// TwinCAT 3 PLC project HOMS_XRT_PLC
// ProjectVersion: 1.0.0
// ProgramVersion: 3.1.4020.4
// libraries:
//   PMPS, * (SLAC - LCLS)
//   Tc2_ControllerToolbox, * (Beckhoff Automation GmbH)
//   Tc2_EtherCAT, * (Beckhoff Automation GmbH)
//   Tc2_MC2, * (Beckhoff Automation GmbH)
//   Tc2_Standard, * (Beckhoff Automation GmbH)
//   Tc2_System, * (Beckhoff Automation GmbH)
//   Tc2_Utilities, * (Beckhoff Automation GmbH)
//   Tc3_Module, * (Beckhoff Automation GmbH)
//   VisuDialogs, * (System)
//   LCLS General,2.4.2,SLAC
//   lcls-twincat-motion,1.4.2,SLAC
//   lcls-twincat-optics,0.1.1,SLAC
//   Tc2_SerialCom,3.3.7.0,Beckhoff Automation GmbH
// project tree:
//   Common/DUTs/ E_GantryControl.TcDUT (not stored), E_GantryMode.TcDUT (not stored), HOMS_Gantry.TcDUT (not stored), HOMS_GantryAxis.TcDUT (not stored), HOMS_PitchMechanismOld.TcDUT (not stored), ST_AbstractAxis.TcDUT (not stored), ST_CoEIndSub.TcDUT (not stored), ST_DecoupledMotionPermits.TcDUT (not stored), ST_ElmoGDCBellCoEParams.TcDUT (not stored), ST_HOMSStepper.TcDUT (not stored), ST_PiezoAxisOld.TcDUT (not stored), ST_StepperStatus.TcDUT (not stored)
//   Common/POUs/Helpers/ FB_Drive.TcPOU (not stored), FB_ElmoGDCBellCoE.TcPOU (not stored), FB_ElmoMCUploadDriveParams.TcPOU (not stored), FB_ElmoStoMonitor.TcPOU (not stored), FB_GantryDiffVirtualLimitSwitch.TcPOU (not stored), FB_InitDriveRefs.TcPOU (not stored), FB_LimitSwitchState.TcPOU (not stored), FB_PitchSoftLimits.TcPOU, FB_PI_E621_SerialDriver.TcPOU (not stored), FB_PI_E621_SerialTransaction.TcPOU (not stored), FB_PTP.TcPOU (not stored), FB_ReadFloatParameter.TcPOU (not stored), FB_ReadParameterInNC.TcPOU (not stored), FB_WriteParameterInNC.TcPOU (not stored), F_PiezoPosition.TcPOU (not stored), MC_SmoothMover.TcPOU (not stored), WithinRange.TcPOU (not stored)
//   Common/POUs/HOMS_FBs/ FB_Gantry.TcPOU (not stored), FB_GantryDifferenceMonitor.TcPOU (not stored), FB_PitchControlOld.TcPOU, FB_ReduceGantryDiff.TcPOU (not stored)
//   / GlobalTextList.TcGTLO (not stored), PiezoDriver.TcTTO (not stored), PlcTask.TcTTO (not stored), SerialIO.TcTTO (not stored), Visualization Manager.TcVMO (not stored)
//   GVLs/ GVL.TcGVL, GVL_COM_Buffers.TcGVL (not stored), GVL_Constants.TcGVL (not stored), GVL_Devices.TcGVL, GVL_IO.TcGVL (not stored), GVL_PMPS.TcGVL (not stored), GVL_SerialIO.TcGVL (not stored), GVL_XRTM1.TcGVL
//   POUs/ FB_MirrorCoatingProtection.TcPOU (not stored), FB_MirrorCoatingProtectionScaledPositions.TcPOU (not stored), FB_MPS_STATES.TcPOU (not stored), Main.TcPOU, PRG_CoatingProtectionScaledPositions.TcPOU (not stored), PRG_CoatingProtection.TcPOU, P_GantryDiffSup.TcPOU (not stored), P_MotionSup.TcPOU (not stored)
//   POUs/Modbus/ p_ModbusRx_OutputCoils.TcPOU (not stored), p_ModbusRx_PLCMemory.TcPOU, p_ModbusTx_InputCoils.TcPOU (not stored), p_ModbusTx_InputReg.TcPOU (not stored), p_ModbusTx_OutputCoils.TcPOU (not stored), p_ModbusTx_PLCMemory.TcPOU
//   POUs/Serial Comm/ PiezoSerial.TcPOU, P_Serial_Com.TcPOU (not stored)
//   VISUs/ GantryControls.TcVIS (not stored), Visualization.TcVIS (not stored), PiezoControls.TcVIS (not stored)
// real-time tasks:
//   TASK PlcTask: cycle T#10ms, priority 20, ADS port 350
//   TASK SerialIO: cycle T#2ms, priority 1, ADS port 351
//   TASK LoggerTask: cycle T#10ms, priority 2, ADS port 352
//   TASK PiezoDriver: cycle T#1ms, priority 3, ADS port 353
// motion (NC):
// I/O:
//   DEVICE HOMS, AmsNetId 172.21.88.136.2.1
//     Term 1 (EK1200) [EK1200-5000 EtherCAT Power supply (2A E-Bus)]
//       Term 24 (EL9187) [EL9187 Potential Connection, 8 x Ground]
//       Term 13 (EL2008) [EL2008 8Ch. Dig. Output 24V, 0.5A]
//       Term 14 (EK1122) [EK1122 2 port EtherCAT junction]
//         EK1100_M1 [EK1100 EtherCAT Coupler (2A E-Bus)]
//           EL7041-1000_M1_Xup [EL7041-1000 1Ch. Stepper motor output stage (50V, 5A, standard)]
//           EL7041-1000_M1_Xdwn [EL7041-1000 1Ch. Stepper motor output stage (50V, 5A, standard)]
//           EL7041-1000_M1_Yup [EL7041-1000 1Ch. Stepper motor output stage (50V, 5A, standard)]
//           EL7041-1000_M1_Ydwn [EL7041-1000 1Ch. Stepper motor output stage (50V, 5A, standard)]
//           EL7041-1000_M1_PitchCoarse [EL7041-1000 1Ch. Stepper motor output stage (50V, 5A, standard)]
//           EL7041-1000_M1_Bender
//           EL6001_M1_PitchFine [EL6001 Interface (RS232)]
//           EL5042_M1_Xupdwn
//           EL5042_M1_Yupdwn
//           EL5042_M1_PitchBender
//           EL1004_M1_STO
//           EL9505_M1_BenderLims
//           Term 42 (EL9011)
//         M2-Y1 (Elmo Drive) [Gold EtherCAT GCON Drive Rev:0x00010420]
//         M2-Y2 (Elmo Drive) [Gold EtherCAT GCON Drive Rev:0x00010420]
//         M2-X1 (Elmo Drive) [Gold EtherCAT GCON Drive Rev:0x00010420]
//         M2-X2 (Elmo Drive) [Gold EtherCAT GCON Drive Rev:0x00010420]
//         M2-P1 (Elmo Drive) [Gold EtherCAT GCON Drive Rev:0x00010420]
//         M2-B1 (Elmo Drive) [Gold EtherCAT GCON Drive Rev:0x00010420]
//         M2-Interface Box (EK1100) [EK1100 EtherCAT Coupler (2A E-Bus)]
//           M2-P1-Piezo (EL6001) [EL6001 Interface (RS232)]
//           M2 (EL9011) [EL9011 End Terminal]
//       Term 2 (EK1122) [EK1122 2 port EtherCAT junction]
//         M3-Y1 (Elmo Drive) [Gold EtherCAT GCON Drive Rev:0x00010420]
//         M3-Y2 (Elmo Drive) [Gold EtherCAT GCON Drive Rev:0x00010420]
//         M3-X1 (Elmo Drive) [Gold EtherCAT GCON Drive Rev:0x00010420]
//         M3-X2 (Elmo Drive) [Gold EtherCAT GCON Drive Rev:0x00010420]
//         M3-P1 (Elmo Drive) [Gold EtherCAT GCON Drive Rev:0x00010420]
//         M3-B1 (Elmo Drive) [Gold EtherCAT GCON Drive Rev:0x00010420]
//         M3-Interface Box (EK1100) [EK1100 EtherCAT Coupler (2A E-Bus)]
//           M3-P1-Piezo (EL6001) [EL6001 Interface (RS232)]
//           M3 (EL9011) [EL9011 End Terminal]
//       Term 34 (EK1521-0010)
// variable links:
//   HOMS_XRT_PLC Instance <-> HOMS
//     PlcTask Inputs/GVL.gAmsNetIDEcatMaster1 <-> InfoData/AmsNetId
//   HOMS_XRT_PLC Instance <-> HOMS/Term 1 (EK1200)/Term 13 (EL2008)
//     PlcTask Outputs/GVL.bXRT_M2_IN <-> Channel 2/Output
//     PlcTask Outputs/GVL.bXRT_M2_OUT <-> Channel 1/Output
//   HOMS_XRT_PLC Instance <-> HOMS/Term 1 (EK1200)/Term 14 (EK1122)/EK1100_M1/EL1004_M1_STO
//     PlcTask Inputs/Main.XRTM1.fbRunHOMS.bSTOEnable1 <-> Channel 1/Input
//     PlcTask Inputs/Main.XRTM1.fbRunHOMS.bSTOEnable2 <-> Channel 2/Input
//   HOMS_XRT_PLC Instance <-> HOMS/Term 1 (EK1200)/Term 14 (EK1122)/EK1100_M1/EL5042_M1_PitchBender
//     PlcTask Inputs/GVL_XRTM1.XRTM1_Pitch.diEncCnt <-> FB Inputs Channel 1/Position
//   HOMS_XRT_PLC Instance <-> HOMS/Term 1 (EK1200)/Term 14 (EK1122)/EK1100_M1/EL5042_M1_Xupdwn
//     PlcTask Inputs/Main.XRTM1.fbRunHOMS.stXdwnEnc/Count <-> FB Inputs Channel 2/Position
//     PlcTask Inputs/Main.XRTM1.fbRunHOMS.stXupEnc/Count <-> FB Inputs Channel 1/Position
//   HOMS_XRT_PLC Instance <-> HOMS/Term 1 (EK1200)/Term 14 (EK1122)/EK1100_M1/EL5042_M1_Yupdwn
//     PlcTask Inputs/Main.XRTM1.fbRunHOMS.stYdwnEnc/Count <-> FB Inputs Channel 2/Position
//     PlcTask Inputs/Main.XRTM1.fbRunHOMS.stYupEnc/Count <-> FB Inputs Channel 1/Position
//   HOMS_XRT_PLC Instance <-> HOMS/Term 1 (EK1200)/Term 14 (EK1122)/EK1100_M1/EL7041-1000_M1_Bender
//     PlcTask Inputs/Main.M6.bLimitBackwardEnable <-> STM Status/Status/Digital input 2
//     PlcTask Inputs/Main.M6.bLimitForwardEnable <-> STM Status/Status/Digital input 1
//   HOMS_XRT_PLC Instance <-> HOMS/Term 1 (EK1200)/Term 14 (EK1122)/EK1100_M1/EL7041-1000_M1_PitchCoarse
//     PlcTask Inputs/Main.M5.bLimitBackwardEnable <-> STM Status/Status/Digital input 2
//     PlcTask Inputs/Main.M5.bLimitForwardEnable <-> STM Status/Status/Digital input 1
//   HOMS_XRT_PLC Instance <-> HOMS/Term 1 (EK1200)/Term 14 (EK1122)/EK1100_M1/EL7041-1000_M1_Xdwn
//     PlcTask Inputs/Main.M4.bLimitBackwardEnable <-> STM Status/Status/Digital input 2
//     PlcTask Inputs/Main.M4.bLimitForwardEnable <-> STM Status/Status/Digital input 1
//   HOMS_XRT_PLC Instance <-> HOMS/Term 1 (EK1200)/Term 14 (EK1122)/EK1100_M1/EL7041-1000_M1_Xup
//     PlcTask Inputs/Main.M3.bLimitBackwardEnable <-> STM Status/Status/Digital input 2
//     PlcTask Inputs/Main.M3.bLimitForwardEnable <-> STM Status/Status/Digital input 1
//   HOMS_XRT_PLC Instance <-> HOMS/Term 1 (EK1200)/Term 14 (EK1122)/EK1100_M1/EL7041-1000_M1_Ydwn
//     PlcTask Inputs/Main.M2.bLimitBackwardEnable <-> STM Status/Status/Digital input 2
//     PlcTask Inputs/Main.M2.bLimitForwardEnable <-> STM Status/Status/Digital input 1
//   HOMS_XRT_PLC Instance <-> HOMS/Term 1 (EK1200)/Term 14 (EK1122)/EK1100_M1/EL7041-1000_M1_Yup
//     PlcTask Inputs/Main.M1.bLimitBackwardEnable <-> STM Status/Status/Digital input 2
//     PlcTask Inputs/Main.M1.bLimitForwardEnable <-> STM Status/Status/Digital input 1
//   HOMS_XRT_PLC Instance <-> HOMS/Term 1 (EK1200)/Term 14 (EK1122)/M2-B1 (Elmo Drive)
//     PlcTask Inputs/GVL_Devices.HOMS2_Bender.stCoE.stPlcDriveRef/nSlaveAddr <-> InfoData/AdsAddr/port
//   HOMS_XRT_PLC Instance <-> HOMS/Term 1 (EK1200)/Term 14 (EK1122)/M2-Interface Box (EK1100)/M2-P1-Piezo (EL6001)
//     SerialIO Inputs/GVL_SerialIO.Serial_P2_stComIn/D[{0..21}] <-> COM Inputs/Data In {0..21}  (22 links)
//     SerialIO Inputs/GVL_SerialIO.Serial_P2_stComIn/Status <-> COM Inputs/Status
//     SerialIO Outputs/GVL_SerialIO.Serial_P2_stComOut/Ctrl <-> COM Outputs/Ctrl
//     SerialIO Outputs/GVL_SerialIO.Serial_P2_stComOut/D[{0..21}] <-> COM Outputs/Data Out {0..21}  (22 links)
//   HOMS_XRT_PLC Instance <-> HOMS/Term 1 (EK1200)/Term 14 (EK1122)/M2-P1 (Elmo Drive)
//     PlcTask Inputs/GVL_Devices.HOMS2_Pitch.Stepper.diInputs <-> Inputs/Digital Inputs
//     PlcTask Inputs/GVL_Devices.HOMS2_Pitch.Stepper.stCoE.stPlcDriveRef/nSlaveAddr <-> InfoData/AdsAddr/port
//     PlcTask Inputs/GVL_Devices.HOMS2_Pitch.diEncCnt <-> Inputs/Position actual value
//   HOMS_XRT_PLC Instance <-> HOMS/Term 1 (EK1200)/Term 14 (EK1122)/M2-X1 (Elmo Drive)
//     PlcTask Inputs/GVL_Devices.HOMS2_XGantry.PAxis.diEncCnt <-> Inputs/Position actual value
//     PlcTask Inputs/GVL_Devices.HOMS2_XGantry.PAxis.diInputs <-> Inputs/Digital Inputs
//     PlcTask Inputs/GVL_Devices.HOMS2_XGantry.PAxis.stCoE.stPlcDriveRef/nSlaveAddr <-> InfoData/AdsAddr/port
//   HOMS_XRT_PLC Instance <-> HOMS/Term 1 (EK1200)/Term 14 (EK1122)/M2-X2 (Elmo Drive)
//     PlcTask Inputs/GVL_Devices.HOMS2_XGantry.SAxis.diInputs <-> Inputs/Digital Inputs
//     PlcTask Inputs/GVL_Devices.HOMS2_XGantry.SAxis.stCoE.stPlcDriveRef/nSlaveAddr <-> InfoData/AdsAddr/port
//   HOMS_XRT_PLC Instance <-> HOMS/Term 1 (EK1200)/Term 14 (EK1122)/M2-Y1 (Elmo Drive)
//     PlcTask Inputs/GVL_Devices.HOMS2_YGantry.PAxis.diEncCnt <-> Inputs/Position actual value
//     PlcTask Inputs/GVL_Devices.HOMS2_YGantry.PAxis.diInputs <-> Inputs/Digital Inputs
//     PlcTask Inputs/GVL_Devices.HOMS2_YGantry.PAxis.stCoE.stPlcDriveRef/nSlaveAddr <-> InfoData/AdsAddr/port
//   HOMS_XRT_PLC Instance <-> HOMS/Term 1 (EK1200)/Term 14 (EK1122)/M2-Y2 (Elmo Drive)
//     PlcTask Inputs/GVL_Devices.HOMS2_YGantry.SAxis.diInputs <-> Inputs/Digital Inputs
//     PlcTask Inputs/GVL_Devices.HOMS2_YGantry.SAxis.stCoE.stPlcDriveRef/nSlaveAddr <-> InfoData/AdsAddr/port
//   HOMS_XRT_PLC Instance <-> HOMS/Term 1 (EK1200)/Term 2 (EK1122)/M3-B1 (Elmo Drive)
//     PlcTask Inputs/GVL_Devices.HOMS3_Bender.stCoE.stPlcDriveRef/nSlaveAddr <-> InfoData/AdsAddr/port
//   HOMS_XRT_PLC Instance <-> HOMS/Term 1 (EK1200)/Term 2 (EK1122)/M3-Interface Box (EK1100)/M3-P1-Piezo (EL6001)
//     SerialIO Inputs/GVL_SerialIO.Serial_P3_stComIn/D[{0..21}] <-> COM Inputs/Data In {0..21}  (22 links)
//     SerialIO Inputs/GVL_SerialIO.Serial_P3_stComIn/Status <-> COM Inputs/Status
//     SerialIO Outputs/GVL_SerialIO.Serial_P3_stComOut/Ctrl <-> COM Outputs/Ctrl
//     SerialIO Outputs/GVL_SerialIO.Serial_P3_stComOut/D[{0..21}] <-> COM Outputs/Data Out {0..21}  (22 links)
//   HOMS_XRT_PLC Instance <-> HOMS/Term 1 (EK1200)/Term 2 (EK1122)/M3-P1 (Elmo Drive)
//     PlcTask Inputs/GVL_Devices.HOMS3_Pitch.Stepper.diInputs <-> Inputs/Digital Inputs
//     PlcTask Inputs/GVL_Devices.HOMS3_Pitch.Stepper.stCoE.stPlcDriveRef/nSlaveAddr <-> InfoData/AdsAddr/port
//     PlcTask Inputs/GVL_Devices.HOMS3_Pitch.diEncCnt <-> Inputs/Position actual value
//   HOMS_XRT_PLC Instance <-> HOMS/Term 1 (EK1200)/Term 2 (EK1122)/M3-X1 (Elmo Drive)
//     PlcTask Inputs/GVL_Devices.HOMS3_XGantry.PAxis.diInputs <-> Inputs/Digital Inputs
//     PlcTask Inputs/GVL_Devices.HOMS3_XGantry.PAxis.stCoE.stPlcDriveRef/nSlaveAddr <-> InfoData/AdsAddr/port
//   HOMS_XRT_PLC Instance <-> HOMS/Term 1 (EK1200)/Term 2 (EK1122)/M3-X2 (Elmo Drive)
//     PlcTask Inputs/GVL_Devices.HOMS3_XGantry.SAxis.diInputs <-> Inputs/Digital Inputs
//     PlcTask Inputs/GVL_Devices.HOMS3_XGantry.SAxis.stCoE.stPlcDriveRef/nSlaveAddr <-> InfoData/AdsAddr/port
//   HOMS_XRT_PLC Instance <-> HOMS/Term 1 (EK1200)/Term 2 (EK1122)/M3-Y1 (Elmo Drive)
//     PlcTask Inputs/GVL_Devices.HOMS3_YGantry.PAxis.diEncCnt <-> Inputs/Position actual value
//     PlcTask Inputs/GVL_Devices.HOMS3_YGantry.PAxis.diInputs <-> Inputs/Digital Inputs
//     PlcTask Inputs/GVL_Devices.HOMS3_YGantry.PAxis.stCoE.stPlcDriveRef/nSlaveAddr <-> InfoData/AdsAddr/port
//   HOMS_XRT_PLC Instance <-> HOMS/Term 1 (EK1200)/Term 2 (EK1122)/M3-Y2 (Elmo Drive)
//     PlcTask Inputs/GVL_Devices.HOMS3_YGantry.SAxis.diInputs <-> Inputs/Digital Inputs
//     PlcTask Inputs/GVL_Devices.HOMS3_YGantry.SAxis.stCoE.stPlcDriveRef/nSlaveAddr <-> InfoData/AdsAddr/port
//   HOMS_XRT_PLC Instance <-> HOMS/Term 1 (EK1200)/Term 34 (EK1521-0010)/Term 23 (EK1501-0010)/PMPS_FFO
//     PlcTask Outputs/GVL_PMPS.g_FastFaultOutput1.q_xFastFaultOut <-> Channel 1/Output
//     PlcTask Outputs/GVL_PMPS.g_FastFaultOutput2.q_xFastFaultOut <-> Channel 2/Output
//   HOMS_XRT_PLC Instance <-> HOMS/Term 1 (EK1200)/Term 34 (EK1521-0010)/Term 23 (EK1501-0010)/PMPS_PRE
//     PlcTask Inputs/PRG_CoatingProtection.fbArbiterIO.i_stCurrentBP <-> IO Inputs/CurrentBP
//     PlcTask Inputs/PRG_CoatingProtection.fbArbiterIO.xTxPDO_state <-> SYNC Inputs/TxPDO state
//     PlcTask Inputs/PRG_CoatingProtection.fbArbiterIO.xTxPDO_toggle <-> SYNC Inputs/TxPDO toggle
//     PlcTask Outputs/GVL_PMPS.g_FastFaultOutput1.q_xFastFaultOut <-> IO Outputs/FFO1
//     PlcTask Outputs/PRG_CoatingProtection.fbArbiterIO.q_stRequestedBP <-> IO Outputs/RequestedBP
//   HOMS_XRT_PLC Instance <-> NC-Task 1 SAF/Axes/M2 B
//     PlcTask Inputs/GVL_Devices.HOMS2_Bender.stAxis.NcToPlc <-> Outputs/ToPlc
//     PlcTask Outputs/GVL_Devices.HOMS2_Bender.stAxis.PlcToNc <-> Inputs/FromPlc
//   HOMS_XRT_PLC Instance <-> NC-Task 1 SAF/Axes/M2 P
//     PlcTask Inputs/GVL_Devices.HOMS2_Pitch.Stepper.stAxis.NcToPlc <-> Outputs/ToPlc
//     PlcTask Outputs/GVL_Devices.HOMS2_Pitch.Stepper.stAxis.PlcToNc <-> Inputs/FromPlc
//   HOMS_XRT_PLC Instance <-> NC-Task 1 SAF/Axes/M2 X1
//     PlcTask Inputs/GVL_Devices.HOMS2_XGantry.PAxis.stAxis.NcToPlc <-> Outputs/ToPlc
//     PlcTask Outputs/GVL_Devices.HOMS2_XGantry.PAxis.stAxis.PlcToNc <-> Inputs/FromPlc
//   HOMS_XRT_PLC Instance <-> NC-Task 1 SAF/Axes/M2 X2
//     PlcTask Inputs/GVL_Devices.HOMS2_XGantry.SAxis.stAxis.NcToPlc <-> Outputs/ToPlc
//     PlcTask Outputs/GVL_Devices.HOMS2_XGantry.SAxis.stAxis.PlcToNc <-> Inputs/FromPlc
//   HOMS_XRT_PLC Instance <-> NC-Task 1 SAF/Axes/M2 Y1
//     PlcTask Inputs/GVL_Devices.HOMS2_YGantry.PAxis.stAxis.NcToPlc <-> Outputs/ToPlc
//     PlcTask Outputs/GVL_Devices.HOMS2_YGantry.PAxis.stAxis.PlcToNc <-> Inputs/FromPlc
//   HOMS_XRT_PLC Instance <-> NC-Task 1 SAF/Axes/M2 Y2
//     PlcTask Inputs/GVL_Devices.HOMS2_YGantry.SAxis.stAxis.NcToPlc <-> Outputs/ToPlc
//     PlcTask Outputs/GVL_Devices.HOMS2_YGantry.SAxis.stAxis.PlcToNc <-> Inputs/FromPlc
//   HOMS_XRT_PLC Instance <-> NC-Task 1 SAF/Axes/M3 B
//     PlcTask Inputs/GVL_Devices.HOMS3_Bender.stAxis.NcToPlc <-> Outputs/ToPlc
//     PlcTask Outputs/GVL_Devices.HOMS3_Bender.stAxis.PlcToNc <-> Inputs/FromPlc
//   HOMS_XRT_PLC Instance <-> NC-Task 1 SAF/Axes/M3 P
//     PlcTask Inputs/GVL_Devices.HOMS3_Pitch.Stepper.stAxis.NcToPlc <-> Outputs/ToPlc
//     PlcTask Outputs/GVL_Devices.HOMS3_Pitch.Stepper.stAxis.PlcToNc <-> Inputs/FromPlc
//   HOMS_XRT_PLC Instance <-> NC-Task 1 SAF/Axes/M3 X1
//     PlcTask Inputs/GVL_Devices.HOMS3_XGantry.PAxis.stAxis.NcToPlc <-> Outputs/ToPlc
//     PlcTask Outputs/GVL_Devices.HOMS3_XGantry.PAxis.stAxis.PlcToNc <-> Inputs/FromPlc
//   HOMS_XRT_PLC Instance <-> NC-Task 1 SAF/Axes/M3 X2
//     PlcTask Inputs/GVL_Devices.HOMS3_XGantry.SAxis.stAxis.NcToPlc <-> Outputs/ToPlc
//     PlcTask Outputs/GVL_Devices.HOMS3_XGantry.SAxis.stAxis.PlcToNc <-> Inputs/FromPlc
//   HOMS_XRT_PLC Instance <-> NC-Task 1 SAF/Axes/M3 Y1
//     PlcTask Inputs/GVL_Devices.HOMS3_YGantry.PAxis.stAxis.NcToPlc <-> Outputs/ToPlc
//     PlcTask Outputs/GVL_Devices.HOMS3_YGantry.PAxis.stAxis.PlcToNc <-> Inputs/FromPlc
//   HOMS_XRT_PLC Instance <-> NC-Task 1 SAF/Axes/M3 Y2
//     PlcTask Inputs/GVL_Devices.HOMS3_YGantry.SAxis.stAxis.NcToPlc <-> Outputs/ToPlc
//     PlcTask Outputs/GVL_Devices.HOMS3_YGantry.SAxis.stAxis.PlcToNc <-> Inputs/FromPlc

// ---- GVLs/GVL.TcGVL
VAR_GLOBAL
	g_psLogHost	: T_IPv4Addr := '172.21.32.9';
	gDefaultSubsystem : E_Subsystem := MOTION;
	gSystemFault	:	BOOL;
	gAmsNetIDEcatMaster1	AT %I* 	: AMSNETID;
	gFirstPass	:	 BOOL := TRUE;
	
	//MPS Outputs
	bXRT_M2_OUT AT %Q* : BOOL:= FALSE;
	bXRT_M2_IN AT %Q* : BOOL:= FALSE;
	
	//Safe-torque-off status
	gM2STO	:	BOOL;
	gM3STO	:	BOOL;
	
	//Global encoder scale
	// For the HOMS, the encoders are all 1nm/cnt which makes things very easy
	gEncScale	:	LREAL := 1;
	
	//Overrides
	////////////////////////////////////
		(* Use at your own risk. These variables may induce unexpected state machine cases,
			and other undesirable effects. They are primarily for testing purposes. Do
		not use them for operations except in the most dire of situations, and with
		full knowledge and understanding of what they do. *)
		gBypassVirtualLimits	:	BOOL;
	
	//ModBus
	/////////////////////////////////////
	/// test mb_Input_Coils[0] with "modpoll -r 32769 -t 1 127.0.0.1" 
	mb_Input_Coils: ARRAY[0..255] OF BOOL;
	/// test mb_Output_Coils[0] with "modpoll -r 32769 -t 0 127.0.0.1" 
	mb_Output_Coils: ARRAY[0..255] OF BOOL;
	/// test mb_Input_Registers[0] with "modpoll -r 32769 -t 3 127.0.0.1" 
	mb_Input_Registers: ARRAY[0..255] OF WORD;
	/// test mb_Output_Registers[0] with "modpoll -r 32769 -t 4 127.0.0.1" 
	mb_Output_Registers: ARRAY[0..255] OF WORD;
	/// test mb_PLC_Memory[0] with "modpoll -r 12289 -t 4 127.0.0.1" 
	mb_PLC_Memory AT %MW0: ARRAY[0..1000] OF WORD;
END_VAR

// ---- GVLs/GVL_Devices.TcGVL
VAR_GLOBAL
	//XRT M1
	HOMS1_Pitch	    :	HOMS_PitchMechanism := (
		ReqPosLimHi := 220,
		ReqPosLimLo := -193,
		diEncPosLimHi := 11216281,
		diEncPosLimLo := 11004512
	);

	//XRT M2
	HOMS2_Pitch	    : HOMS_PitchMechanism := (
		ReqPosLimHi := 960,
		ReqPosLimLo := -967,
		diEncPosLimHi := 10317713,
		diEncPosLimLo := 9329162
	);
	HOMS2_YGantry	: HOMS_Gantry;
	HOMS2_XGantry	: HOMS_Gantry;
	HOMS2_Bender	:	ST_HOMSStepper;
	
	//XRT M3
	HOMS3_Pitch	    : HOMS_PitchMechanism := (
		ReqPosLimHi := 246,
		ReqPosLimLo := -212,
		diEncPosLimHi := 9123828,
		diEncPosLimLo := 8888874
	);
	HOMS3_YGantry	: HOMS_Gantry;
	HOMS3_XGantry	: HOMS_Gantry;
	HOMS3_Bender	:	ST_HOMSStepper;
	
END_VAR

// ---- GVLs/GVL_XRTM1.TcGVL
{attribute 'qualified_only'}
VAR_GLOBAL
	//XRT M1
	{attribute 'TcLinkTo' := '.diEncCnt:=TIIB[EL5042_M1_PitchBender]^FB Inputs Channel 1^Position'}
	XRTM1_Pitch	    :	HOMS_PitchMechanism := (
		ReqPosLimHi := 220,
		ReqPosLimLo := -193,
		diEncPosLimHi := 11216281,
		diEncPosLimLo := 11004512
	);
END_VAR

// ---- Common/POUs/Helpers/FB_PitchSoftLimits.TcPOU
FUNCTION_BLOCK FB_PitchSoftLimits
VAR_INPUT
	Pitch	:	HOMS_PitchMechanismOld;
END_VAR
VAR_OUTPUT
	xHiLS	:	BOOL;
	xLoLS	:	BOOL;
END_VAR
VAR
	diHys	:	DINT := 500; //500 nm (1 inc/nm)
	STO: BOOL;
END_VAR

STO := Pitch.Stepper.diInputs.3;

xHiLS S= Pitch.diEncCnt < Pitch.diEncPosLimHi - diHys;
xHiLS R= Pitch.diEncCnt > Pitch.diEncPosLimHi;

xLoLS S= Pitch.diEncCnt > Pitch.diEncPosLimLo + diHys;
xLoLS R= Pitch.diEncCnt < Pitch.diEncPosLimLo;

xHiLS := xHiLS AND STO;
xLoLS := xLoLS AND STO;

END_FUNCTION_BLOCK

// ---- Common/POUs/HOMS_FBs/FB_PitchControlOld.TcPOU
{attribute 'reflection'}
FUNCTION_BLOCK FB_PitchControlOld
VAR_IN_OUT
	Pitch : HOMS_PitchMechanismOld;
END_VAR
VAR_INPUT
	DirectPiezoMode	:	BOOL := FALSE; //Set this true to tell the piezo what position to seek in closed loop
	rReqAbsPos	:	REAL; //Control the pitch position with this when DirectPiezoMode is false
END_VAR
VAR_OUTPUT
	q_xError	:	BOOL;
	q_xDone	:	BOOL;
	q_xBusy	:	BOOL;
END_VAR
VAR
	//Introspection
	//////////////////////////////
		{attribute 'instance-path'}
		{attribute 'no_init'}
		POUName	:	STRING; //Name of the POU for logging/error reporting
	
	
	//FB Boilerplate
	//////////////////////
		stDiag	:	ST_fbDiagnostics;
		fbFormatString	:	FB_FormatString;
		
	//Working variables
	/////////////////////////
		PC_State 		:	E_PitchControl := PCM_Init;
		rPrevReqAbsPos	:	REAL; //Previously  requested abs position
		rPrevStepperPos :	REAL; //Previously successfully achieved stepper position
		tonStepperHold	:	TON := (PT := T#100MS); //Timer to hold stepper position while the system relaxes
		FirstPass	:	BOOL := TRUE; //set false after first pass, used for initializations
		Coarse50PiezoMove	:	BOOL;
		OriginalPosRequest: REAL;
		//PTP
		/////////////////////////
				Drive         : FB_DRIVE;
				fbCoE         : FB_ElmoGDCBellCoE;
				nCommand      : UINT;
				rLastSetpoint : REAL;
				rtTweakFwd    : R_TRIG;
				rtTweakBwd    : R_TRIG;
				rtExecute     : R_TRIG;
				bRequesting   : BOOL;
				rSetpoint     : REAL; //Adjusted based on abs pos request or tweaks.
				mcSmoothMover	:	MC_SmoothMover;
	
	//Axis Control Blocks
	/////////////////////////////
		fbPiezoControl	:	FB_PiezoControl;
	
	
	//Triggers
	//////////////////////////////
		rtManualMode:	R_TRIG;
		ftManualMode	:	F_TRIG;
		rtStepperDone	:	R_TRIG;

	lrActPos: LREAL;
	tonPiezoSettled	: TON := (PT:=T#2S);
	tonPiezoDone	:	TON := (PT:=T#500ms);
	
	ftLimitSwitch: F_TRIG;
	// Flag to track when a limit switch has been hit.
	xLimitHit: BOOL;
	rtPiezoMoveDone: R_TRIG;
	rtHalt: R_TRIG;
	bCoarseMoveComplete	:	BOOL; //Set after a coarse move completes, added because coarse moves can be interrupted
END_VAR
VAR CONSTANT
	cPiezoRange	:	REAL := 60; // 90um of stroke to the piezo, which means a 180urad stroke...
    cOperatingRegion : REAL := 0.75; // Only use a fraction of the piezo range before forcing a coarse move    
END_VAR

(* HOMS Pitch Control
A. Wallace

The HOMS Pitch mechanism consists of a stepper and piezo that work together to adjust
the pitch of the mirror assembly.

Pitch control state machine

If the target position is beyond the range of the piezo mechanism,
execute a coarse pitch move with the stepper. 
The target of the coarse move shall be set to the requested position. 
Once coarse motion has completed the coarse motion drive position 
correction output shall be set to zero.

Fine pitch motion with the piezo will be initiated to finish closing the loop.

The piezo mechanism can actuate ~ 180urad or 90um.

*)

lrActPos := Pitch.Stepper.stAxis.NcToPlc.ActPos;
nCommand  := 3;
(* If we hit a limit during a move, we need to change the setpoint *)
ftLimitSwitch(CLK:=Pitch.Stepper.xHiLS AND Pitch.Stepper.xLoLS);

//Manual mode switching logic
/////////////////////////////////////
	rtManualMode(CLK:=DirectPiezoMode);
	ftManualMode(CLK:=DirectPiezoMode);
	A_ModeSwitch();

//Motion control logic from PTP	
//Tweak Triggers
/////////////////////////////////////////////
	rtTweakFwd(CLK:=Pitch.Axis.bTwkFwd);
	rtTweakBwd(CLK:=Pitch.Axis.bTwkBwd);
	rtExecute(CLK:=NOT Pitch.Stepper.stAxis.Status.NotMoving);
	
//Tweak Forward
/////////////////////
IF rtTweakFwd.Q THEN
	//Setup move
	Pitch.Axis.rReqAbsPos := rLastSetpoint + Pitch.Axis.rTweak;
//Tweak Backwards
/////////////////////
ELSIF rtTweakBwd.Q THEN
	//Setup move
	Pitch.Axis.rReqAbsPos := rLastSetpoint - Pitch.Axis.rTweak;
ELSE
	bRequesting := FALSE;
END_IF

(* At this point, Pitch.Axis.rReqAbsPos holds the next setpoint.
Now it will be validated against the soft-limits
*)

//Halt
///////////////////////////////////
	rtHalt(CLK:= Pitch.Axis.xStop);
	(* Halt does the following
	Halts stepper motion, waits for stepper to settle, records stepper position as prev. stepper pos.
	moves to fine move with a new abs setpoint
	*)
	IF rtHalt.Q AND NOT q_xDone THEN
		PC_State := PCM_Halt;
	END_IF

//Check for new position requests, and sanitize
///////////////////////////////////////////////
	IF (rLastSetpoint <> Pitch.Axis.rReqAbsPos) THEN
		//We don't want to initiate any kind of a move if we don't have to.
		IF 	Pitch.Axis.rReqAbsPos > Pitch.ReqPosLimHi OR Pitch.Axis.rReqAbsPos < Pitch.ReqPosLimLo OR
			(Pitch.Axis.rReqAbsPos < lrActPos) AND Pitch.Axis.xLoLS OR (Pitch.Axis.rReqAbsPos > lrActPos) AND Pitch.Axis.xHiLS THEN
			//Requested move is outside of travel limits
			OriginalPosRequest	:= Pitch.Axis.rReqAbsPos;
			Pitch.Axis.rReqAbsPos := LIMIT(Pitch.ReqPosLimLo, Pitch.Axis.rReqAbsPos, Pitch.ReqPosLimHi);
			//Only want to log one warning about a bad position request.
			IF OriginalPosRequest <> Pitch.Axis.rReqAbsPos THEN
				//Log a warning
				fbFormatString.sFormat := 'Pitch req OoR fb (%s), reset within limits, %f';
				fbFormatString.arg1 := F_STRING(POUName);
				fbFormatString.arg2 := F_REAL(OriginalPosRequest);
				//fbFormatString(sOut=>fbLogMessage.i_sMsg);
				fbFormatString(sOut=>stDiag.asResults[stDiag.resultIdx.IncVal()]);
				//fbLogMessage(i_eSevr:= Warning, i_eSubsystem:=gDefaultSubsystem);
			END_IF
		END_IF
		// At this point Pitch.Axis.rReqAbsPos is considered clean and safe, so we pass to a holding variable
		rSetpoint := Pitch.Axis.rReqAbsPos;
		//Set the previously requested position here
		rLastSetpoint := rSetpoint;
		//New position request, no longer done.
		q_xDone := FALSE;
		q_xBusy	:= TRUE;
		PC_State := PCM_MoveRequested;
	END_IF
	
//State Machine
//////////////////////////////////
CASE PC_State OF
	PCM_Init: 
		//Initialize stepper motor mc power block
		Drive.bReset := FirstPass;
		PC_State := PCM_Standby;
		
	PCM_Standby:
		;
		
	PCM_MoveRequested: 
		//A move has been requested, is it within range of the piezo?
		IF WithinRange(ValA:=rSetpoint, Center:=rPrevStepperPos, Range:=cPiezoRange, Offset:=0)
                //Ensure that the piezo is not currently outside the operating range
                //Otherwise, force a coarse move that will rezero the piezo travel
	        AND WithinRange(ValA:=Pitch.Piezo.rActVoltage,
                                Center:=(Pitch.Piezo.LowerVoltage + Pitch.Piezo.UpperVoltage)/2.0,
                                Range:=cOperatingRegion*(Pitch.Piezo.UpperVoltage - Pitch.Piezo.LowerVoltage)/2.0,
                                Offset:=0)
			AND bCoarseMoveComplete
		THEN
			//Move is within the nominal range of the piezo
			fbFormatString.sFormat := 'Within range, fine move %f';
			fbFormatString.arg1 := F_REAL(rSetpoint);
			fbFormatString(sOut=>stDiag.asResults[stDiag.resultIdx.IncVal()]);
			PC_State := PCM_FineMove;
		ELSE
			// Out of range, head to coarse move
			fbFormatString.sFormat := 'OoR, using stepper %f';
			fbFormatString.arg1 := F_REAL(rSetpoint);
			fbFormatString(sOut=>stDiag.asResults[stDiag.resultIdx.IncVal()]);
			bCoarseMoveComplete := FALSE;
			PC_State := PCM_Coarse50Piezo;
		END_IF
		
	PCM_Coarse50Piezo:
		//A coarse move uses the stepper to do a best-effort position
		//First set the piezo to nominal 50% extension using idle mode
		//////////////////////////////////////////////////////////////////////////////
		Pitch.Piezo.xIdleMode := TRUE;
		//Indicate we are doing the coarse 50% piezo move	
		Coarse50PiezoMove := TRUE;
		//Wait for piezo to settle
		tonPiezoSettled.IN := TRUE;
		Coarse50PiezoMove R= tonPiezoSettled.Q;
		IF tonPiezoSettled.Q THEN
			//Piezo has moved to 50% position, finish with the stepper
			PC_State := PCM_CoarseMove;
			Pitch.Stepper.xEnable := TRUE;
			tonPiezoSettled.IN := FALSE;
		END_IF
		
	PCM_CoarseMove: 
		//With the piezo at a nom 50% extension, move the stepper to requested position
		IF Drive.bEnabled THEN
			//Drive.fPosition := rSetpoint;
			//Drive.bExecute := TRUE;
			
			mcSmoothMover.ReqAbsPos := rSetpoint;
			mcSmoothMover.Enable := TRUE;
		END_IF

		IF ftLimitSwitch.Q THEN
			Drive.fPosition := lrActPos;
			
			mcSmoothMover.ReqAbsPos := lrActPos;
			
			xLimitHit	:= TRUE; //set this flag here.
		END_IF
		tonStepperHold.IN := WithinRange(ValA:=LREAL_TO_REAL(lrActPos), Center:=rSetpoint, Range:=Pitch.Stepper.rStepperDmovRange, Offset:=0);
		tonStepperHold(); //call this here to reset Q just below on first cycle
		//If the coarse move is complete, finish position correction with the piezo
		IF tonStepperHold.Q  OR ftLimitSwitch.Q THEN
			PC_State := PCM_CoarseMoveCleanup;
		ELSIF Pitch.Stepper.stStatus.bError OR Drive.bError OR mcSmoothMover.Error THEN
			Drive.bExecute := FALSE;
			mcSmoothMover.Enable := FALSE;
			Pitch.Stepper.xEnable := FALSE;
			PC_State := PCM_StepperError;
			//Stepper fb has encountered an error, pass a message to the logger
			IF Pitch.Stepper.stStatus.bError THEN
				fbFormatString.sFormat := 'Coarse move error, stepper err id %d';
				fbFormatString.arg1 := F_UDINT(Pitch.Stepper.stStatus.nErrorId);
			ELSIF Drive.bError THEN
				fbFormatString.sFormat := 'Coarse move error, drive err id %d';
				fbFormatString.arg1 := F_UDINT(Drive.nErrorId);
			ELSIF mcSmoothMover.Error THEN
				fbFormatString.sFormat := 'Coarse move error, smoothmover error';
			END_IF
			fbFormatString(sOut=>stDiag.asResults[stDiag.resultIdx.IncVal()]);
		END_IF
		
	PCM_CoarseMoveCleanup:
		Drive.bExecute := FALSE;
		//Calling Drive with execute false will halt the axis
		//Once halted, the axis will be in standstill
		// then we can disble it without error.
		IF Pitch.Stepper.stAxis.Status.StandStill THEN
			Pitch.Stepper.xEnable := FALSE;
		END_IF
		IF Pitch.Stepper.stAxis.Status.Disabled THEN
			rPrevStepperPos := mcSmoothMover.ReqAbsPos;
			bCoarseMoveComplete	:= TRUE;
			PC_State := PCM_FineMove;
		END_IF

	PCM_FineMove:	
		Pitch.Piezo.xIdleMode := FALSE;
		fbPiezoControl.xExecute := TRUE;
		IF xLimitHit THEN
			Pitch.Piezo.rReqAbsPos := lrActPos;
		ELSE
			Pitch.Piezo.rReqAbsPos := rSetpoint;
		END_IF
		rtPiezoMoveDone(CLK:=fbPiezoControl.xDone);
		IF rtPiezoMoveDone.Q THEN
			fbPiezoControl.xExecute := FALSE;
			PC_State := PCM_Done;
		END_IF
		
	PCM_Halt:
		//We may transition to this state from anywhere, so we need to clean up and move to done
		//Halt the stepper
		//If trans. from FineMove, stepper is already disabled
		Drive.bExecute := FALSE;
		IF Pitch.Stepper.stAxis.Status.Standstill OR Pitch.Stepper.stAxis.Status.Disabled THEN
			Pitch.Stepper.xEnable := FALSE;
			//If the piezo control is done, we haven't started the fine move yet, so we can
			// record the current position as the prev. achv. stepper position.
			IF fbPiezoControl.xDone THEN
				rPrevStepperPos := lrActPos;
			END_IF
			// Very special case, where the setpoint is now where we halted
			rSetpoint := lrActPos;
			PC_State := PCM_FineMove;
		END_IF
		
	PCM_Done:
		
		Pitch.Axis.rReqAbsPos := rLastSetpoint; //this might be kind of funky
		xLimitHit := FALSE;
		//Indicate we're done
		q_xDone	:= TRUE;
		q_xBusy := FALSE;
		//Move back to standby
		PC_State := PCM_Standby;
	PCM_StepperError:
		Drive.bReset := TRUE; // set false again in PCM_Init
		q_xBusy := FALSE;
		PC_State := PCM_Init; 
	PCM_PiezoError:
		q_xBusy := FALSE;
		PC_State := PCM_Init;
	PCM_OtherError:
		q_xBusy := FALSE;
		PC_State := PCM_Init;
	
END_CASE

FirstPass := FALSE;

//Transfer the other stuff to the piezo
/////////////////////////////////////////
Pitch.Piezo.rActPos := lrActPos;

//Function blocks
ACT_PTP();

tonPiezoSettled();
tonStepperHold();

fbPiezoControl(iq_Piezo:=Pitch.Piezo,
	Enable_Positive:=Pitch.Stepper.xHiLS,
	Enable_Negative:=Pitch.Stepper.xLoLS
);

ACTION A_ModeSwitch:
(* When switching between modes, we need to make sure all the executes/ mode switches, etc. are cleared *)

// Automatic to manual
/////////////////////////////
IF rtManualMode.Q THEN
;
END_IF

// Manual to automatic
//////////////////////////////
IF ftManualMode.Q THEN
	;
END_IF
END_ACTION

ACTION ACT_PTP:
//Read CoE Parameters
/////////////////////////
fbCoE(stCoE:=Pitch.Stepper.stCoE);

//Give control of the axis to the Drive function block
///////////////////////////////////////////////////////
Drive(bEnable  := Pitch.Stepper.xEnable,
	  Axis     := Pitch.Stepper.stAxis,
	  nCommand := nCommand,
	  fAcceleration := Pitch.Stepper.fAcceleration,
	  fDeceleration := Pitch.Stepper.fDeceleration,
	  fVelocity     := Pitch.Stepper.fVelocity,
	  bLimitFwd     := Pitch.Stepper.xHiLS,
	  bLimitBwd     := Pitch.Stepper.xLoLS,
	  bDone	=>  Pitch.Stepper.bDone,
	  bBusy => Pitch.Stepper.bBusy,
	  stStepperStatus => Pitch.Stepper.stStatus
	  );

//Reset Execute to wait for next motion command
////////////////////////////////////////////////
//bExecute R= Drive.Status.NotMoving AND NOT bRequesting;

//MC Smooth Mover
////////////////////////////////////////////////
(* You can control an axis with MC blocks other than those in PTP or drive.
We just use the drive/PTP block to initialize the axis and manage the limit
switch logic *)
mcSmoothMover(Axis:=Pitch.Stepper.stAxis,
	Velocity:=Pitch.Stepper.fVelocity);
END_ACTION

END_FUNCTION_BLOCK

// ---- POUs/Main.TcPOU
PROGRAM Main
VAR
	// Beckhoff Version of XRT-M1
	// XRTM1
	// Motors
	{attribute 'TcLinkTo' := '.bLimitForwardEnable:=TIIB[EL7041-1000_M1_Yup]^STM Status^Status^Digital input 1;
                              .bLimitBackwardEnable:=TIIB[EL7041-1000_M1_Yup]^STM Status^Status^Digital input 2'}
	{attribute 'pytmc' := '
		pv: XRTM1:HOMS:MMS:YUP
	'}
	M1 : DUT_MotionStage := (fVelocity:=200.0, nEnableMode:=ENUM_StageEnableMode.ALWAYS, bPowerSelf:=TRUE); // XRT-M1 Yup
	fbMotionStage_m1 : FB_MotionStage;

	{attribute 'TcLinkTo' := '.bLimitForwardEnable:=TIIB[EL7041-1000_M1_Ydwn]^STM Status^Status^Digital input 1;
                              .bLimitBackwardEnable:=TIIB[EL7041-1000_M1_Ydwn]^STM Status^Status^Digital input 2'}
	{attribute 'pytmc' := '
		pv: XRTM1:HOMS:MMS:YDWN
	'}
	M2 : DUT_MotionStage := (fVelocity:=200.0, nEnableMode:=ENUM_StageEnableMode.ALWAYS, bPowerSelf:=TRUE); // XRT-M1 Ydwn
	fbMotionStage_m2 : FB_MotionStage;

	{attribute 'TcLinkTo' := '.bLimitForwardEnable:=TIIB[EL7041-1000_M1_Xup]^STM Status^Status^Digital input 1;
                              .bLimitBackwardEnable:=TIIB[EL7041-1000_M1_Xup]^STM Status^Status^Digital input 2'}
	{attribute 'pytmc' := '
		pv: XRTM1:HOMS:MMS:XUP
	'}
	M3 : DUT_MotionStage := (fVelocity:=1000.0, nEnableMode:=ENUM_StageEnableMode.ALWAYS, bPowerSelf:=TRUE); // XRT-M1 Xup
	fbMotionStage_m3 : FB_MotionStage;

	{attribute 'TcLinkTo' := '.bLimitForwardEnable:=TIIB[EL7041-1000_M1_Xdwn]^STM Status^Status^Digital input 1;
                              .bLimitBackwardEnable:=TIIB[EL7041-1000_M1_Xdwn]^STM Status^Status^Digital input 2'}
	{attribute 'pytmc' := '
		pv: XRTM1:HOMS:MMS:XDWN
	'}
	M4 : DUT_MotionStage := (fVelocity:=1000.0, nEnableMode:=ENUM_StageEnableMode.ALWAYS, bPowerSelf:=TRUE); // XRT-M1 Xdwn
	fbMotionStage_m4 : FB_MotionStage;

	{attribute 'TcLinkTo' := '.bLimitForwardEnable:=TIIB[EL7041-1000_M1_PitchCoarse]^STM Status^Status^Digital input 1;
                              .bLimitBackwardEnable:=TIIB[EL7041-1000_M1_PitchCoarse]^STM Status^Status^Digital input 2'}
	{attribute 'pytmc' := '
		pv: XRTM1:HOMS:MMS:PITCH
	'}
	M5 : DUT_MotionStage := (fVelocity:=150.0); // XRT-M1 Pitch Stepper

	{attribute 'TcLinkTo' := '.bLimitForwardEnable:=TIIB[EL7041-1000_M1_Bender]^STM Status^Status^Digital input 1;
                              .bLimitBackwardEnable:=TIIB[EL7041-1000_M1_Bender]^STM Status^Status^Digital input 2'}
	{attribute 'pytmc' := '
		pv: XRTM1:HOMS:MMS:BENDER
	'}
	M6 : DUT_MotionStage := (fVelocity:=150.0, nEnableMode:=ENUM_StageEnableMode.ALWAYS, bPowerSelf:=TRUE); // XRT-M1 Bender
	fbMotionStage_m6 : FB_MotionStage;

	{attribute 'TcLinkTo' := '.fbRunHOMS.bSTOEnable1:=TIIB[EL1004_M1_STO]^Channel 1^Input;
                              .fbRunHOMS.bSTOEnable2:=TIIB[EL1004_M1_STO]^Channel 2^Input;
	                          .fbRunHOMS.stYupEnc.Count:=TIIB[EL5042_M1_Yupdwn]^FB Inputs Channel 1^Position;
	                          .fbRunHOMS.stYdwnEnc.Count:=TIIB[EL5042_M1_Yupdwn]^FB Inputs Channel 2^Position;
	                          .fbRunHOMS.stXupEnc.Count:=TIIB[EL5042_M1_Xupdwn]^FB Inputs Channel 1^Position;
	                          .fbRunHOMS.stXdwnEnc.Count:=TIIB[EL5042_M1_Xupdwn]^FB Inputs Channel 2^Position'}
	{attribute 'pytmc' := '
		pv: XRTM1:HOMS
	'}
	XRTM1 : DUT_HOMS;

	// Encoder Arrays/RMS Watch:
	{attribute 'pytmc' := '
		pv: XRTM1:HOMS:ENC:Y
	'}
	fbYRMSErrorXRTM1 : FB_RMSWatch;
	fMaxYRMSErrorXRTM1 : LREAL;
	fMinYRMSErrorXRTM1 : LREAL;

	{attribute 'pytmc' := '
		pv: XRTM1:HOMS:ENC:X
	'}
	fbXRMSErrorXRTM1 : FB_RMSWatch;
	fMaxXRMSErrorXRTM1 : LREAL;
	fMinXRMSErrorXRTM1 : LREAL;

	{attribute 'pytmc' := '
		pv: XRTM1:HOMS:ENC:PITCH
	'}
	fbPitchRMSErrorXRTM1 : FB_RMSWatch;
	fMaxPitchRMSErrorXRTM1 : LREAL;
	fMinPitchRMSErrorXRTM1 : LREAL;

	{attribute 'pytmc' := '
		pv: XRTM1:HOMS:ENC:BENDER
	'}
	fbBenderRMSErrorXRTM1 : FB_RMSWatch;
	fMaxBenderRMSErrorXRTM1 : LREAL;
	fMinBenderRMSErrorXRTM1 : LREAL;

	// Pitch Control
	fbXRTM1PitchControl : FB_PitchControl;
	bXRTM1PitchDone : BOOL;
	bXRTM1PitchBusy : BOOL;

	// Bender Control
	fbBenderXRTM1 : FB_Bender;

	// Raw Encoder Counts
	{attribute 'pytmc' := '
		pv: XRTM1:HOMS:ENC:YUP:CNT
		field: EGU cnt
		io: i
	'}
	nEncCntYupXRTM1 : UDINT;
	{attribute 'pytmc' := '
		pv: XRTM1:HOMS:ENC:YDWN:CNT
		field: EGU cnt
		io: i
	'}
	nEncCntYdwnXRTM1 : UDINT;
	{attribute 'pytmc' := '
		pv: XRTM1:HOMS:ENC:XUP:CNT
		field: EGU cnt
		io: i
	'}
	nEncCntXupXRTM1 : UDINT;
	{attribute 'pytmc' := '
		pv: XRTM1:HOMS:ENC:XDWN:CNT
		field: EGU cnt
		io: i
	'}
	nEncCntXdwnXRTM1 : UDINT;
	{attribute 'pytmc' := '
		pv: XRTM1:HOMS:ENC:PITCH:CNT
		field: EGU cnt
		io: i
	'}
	nEncCntPitchXRTM1 : UDINT;

	// Encoder Reference Values
	{attribute 'pytmc' := '
		pv: XRTM1:HOMS:ENC:YUP:REF
		field: EGU cnt
		io: i
	'}
	nEncRefYupXRTM1 : UDINT;
	{attribute 'pytmc' := '
		pv: XRTM1:HOMS:ENC:YDWN:REF
		field: EGU cnt
		io: i
	'}
	nEncRefYdwnXRTM1 : UDINT;
	{attribute 'pytmc' := '
		pv: XRTM1:HOMS:ENC:XUP:REF
		field: EGU cnt
		io: i
	'}
	nEncRefXupXRTM1 : UDINT;
	{attribute 'pytmc' := '
		pv: XRTM1:HOMS:ENC:XDWN:REF
		field: EGU cnt
		io: i
	'}
	nEncRefXdwnXRTM1 : UDINT;
	{attribute 'pytmc' := '
		pv: XRTM1:HOMS:ENC:PITCH:REF
		field: EGU cnt
		io: i
	'}
	nEncRefPitchXRTM1 : UDINT;
	mcReadParameterPitchXRTM1 : MC_ReadParameter;
	fEncRefPitchXRTM1_urad : LREAL; // Current Pitch encoder offset in urad
	///////////////////////////////////////////////////////////////////////

	tpImAPLC : TP := (PT:=T#10S);

	XRTM2PitchControl	    :	FB_PitchControlOld;
	//{attribute 'TcLinkTo' := 	'.Gantry.diEncCnt	:=	TIIB[M2-Y1 (Elmo Drive)]^Inputs^Position actual value'}
	XRTM2Y_GantryControl	:	FB_Gantry;
	XRTM2X_GantryControl	:	FB_Gantry;
	XRTM3PitchControl	    :	FB_PitchControlOld;
//	{attribute 'TcLinkTo' := 	'.Gantry.diEncCnt	:=	TIIB[M3-Y1 (Elmo Drive)]^Inputs^Position actual value'}
	XRTM3Y_GantryControl	:	FB_Gantry;
	XRTM3X_GantryControl	:	FB_Gantry;
	
	
	// Expert mode permits direct access to individual acutators.
	ExpertMode	:	BOOL := FALSE;
	PitchManualMode: BOOL := FALSE;
	
	//Limit switch evaluation blocks
	fbM2Y1LS	:	FB_LimitSwitchState;
	fbM2Y2LS	:	FB_LimitSwitchState;
	fbM2X1LS	:	FB_LimitSwitchState;
	fbM2X2LS	:	FB_LimitSwitchState;
	fbM2P1LS	:	FB_PitchSoftLimits;	
	
	fbM3Y1LS	:	FB_LimitSwitchState;
	fbM3Y2LS	:	FB_LimitSwitchState;
	fbM3X1LS	:	FB_LimitSwitchState;
	fbM3X2LS	:	FB_LimitSwitchState;
	fbM3P1LS	:	FB_PitchSoftLimits;	
	
	//Drive CoE Fb
	fbY1CoE	:	FB_ElmoGDCBellCoE;
	fbY2CoE	:	FB_ElmoGDCBellCoE;
	
	fbX1CoE	:	FB_ElmoGDCBellCoE;
	fbX2CoE	:	FB_ElmoGDCBellCoE;
	
	fbP1CoE	:	FB_ElmoGDCBellCoE;
	fbB1CoE	:	FB_ElmoGDCBellCoE;
	
	
	//Init params trigger
	rtInitParams	:	R_TRIG;
	
	//Test Parameters
		rStepSize: REAL;
	SettleTime: TON := (
	PT:=T#2s);
	TestUpperVoltage: REAL := 100;
	TestLowerVoltage: REAL := 10;
	xRunPiezoRepeatTest: BOOL;
	
	//Drive reference initializations
	fbInitDriveRef	:	FB_InitDriveRefs;
	//MPS Information
	fbMPS_States :  FB_MPS_STATES;
	M2_INRANGE  :   ARRAY[0..1] OF DINT := [24568920, 26568920];
	M2_OUTRANGE  :  ARRAY[0..1] OF DINT := [43568250, 50570250];
	//noConsequence	:	BOOL;
	
	mcBenderPower	:	MC_POWER;
	
	// Logging
	fbLogHandler : FB_LogHandler;
END_VAR

// Beckhoff Version of XRT-M1
// Raw Encoder Counts For Epics
nEncCntYupXRTM1 := ULINT_TO_UDINT(XRTM1.fbRunHOMS.stYupEnc.Count);
nEncCntYdwnXRTM1 := ULINT_TO_UDINT(XRTM1.fbRunHOMS.stYdwnEnc.Count);
nEncCntXupXRTM1 := ULINT_TO_UDINT(XRTM1.fbRunHOMS.stXupEnc.Count);
nEncCntXdwnXRTM1 := ULINT_TO_UDINT(XRTM1.fbRunHOMS.stXdwnEnc.Count);
nEncCntPitchXRTM1 := LINT_TO_UDINT(GVL_XRTM1.XRTM1_Pitch.diEncCnt);
//////////////////////////////////////////////////////////////
//System IO
/////////////////////////////
p_ModbusRx_OutputCoils();
p_ModbusRx_PLCMemory();


//InitParams
////////////////////
rtInitParams(CLK:=gFirstPass);
IF rtInitParams.Q THEN
	Init_XRTM2();
	Init_XRTM3();
	gFirstPass := FALSE;
END_IF

//System Error Handling
/////////////////////////////////////
//SystemErrorSummary(); //Check this action for a summary of all system faults
					  
//SystemError();

//Driver Parameter Verification
/////////////////////////////////////

//Gantry Interlock Logic
/////////////////////////////////////
	//SimGantry.VAxis.i_xMotorInterlock := TRUE;
	//SimGantry.PAxis.i_xMotorInterlock := TRUE;
	//SimGantry.SAxis.i_xMotorInterlock := TRUE;

LimitSwitchIO();
	
// Pitch control
/////////////////////////////////////
XRTM2PitchControl(Pitch:=HOMS2_Pitch, DirectPiezoMode:=(ExpertMode AND PitchManualMode), q_xDone=>HOMS2_Pitch.Axis.bDone, q_xBusy => HOMS2_Pitch.Axis.bBusy);
XRTM3PitchControl(Pitch:=HOMS3_Pitch, DirectPiezoMode:=(ExpertMode AND PitchManualMode), q_xDone=>HOMS3_Pitch.Axis.bDone, q_xBusy => HOMS3_Pitch.Axis.bBusy);

//Y motion
/////////////////////////////////////
XRTM2Y_GantryControl(Gantry:=HOMS2_YGantry);
XRTM3Y_GantryControl(Gantry:=HOMS3_YGantry);

HOMS3_YGantry.PAxis.stAxis.ReadStatus();
HOMS3_YGantry.SAxis.stAxis.ReadStatus();
HOMS3_YGantry.PAxis.stStatus.rActPosition := LREAL_TO_REAL(HOMS3_YGantry.PAxis.stAxis.NcToPlc.ActPos);
HOMS3_YGantry.SAxis.stStatus.rActPosition := LREAL_TO_REAL(HOMS3_YGantry.SAxis.stAxis.NcToPlc.ActPos);
	
//X Motion
/////////////////////////////////////
XRTM2X_GantryControl(Gantry:=HOMS2_XGantry);
XRTM3X_GantryControl(Gantry:=HOMS3_XGantry);

//Communicate state to MPS
////////////////////////////////
fbMPS_States(GANTRY:=HOMS2_XGantry,
			 OUT_LS:=NOT HOMS2_XGantry.PAxis.xHiLS OR NOT HOMS2_XGantry.SAxis.xLoLS,
			 IN_RANGE:=M2_INRANGE,
			 OUT_RANGE:=M2_OUTRANGE);
			 
bXRT_M2_IN  := fbMPS_States.IN;
bXRT_M2_OUT := fbMPS_States.OUT;

//EPICS Tx Update
////////////////////
p_ModbusTx_InputCoils();
//p_ModbusTx_OutputCoils();
p_ModbusTx_InputReg();
p_ModbusTx_PLCMemory();

//PMPS
PRG_CoatingProtection();

// Logging
fbLogHandler();

ACTION Init_XRTM2:
//FEE-M2
///////////////////////////


//Initialize ELMO Drive references
fbInitDriveRef(stCoE:=HOMS2_XGantry.PAxis.stCoE);
fbInitDriveRef(stCoE:=HOMS2_XGantry.SAxis.stCoE);
fbInitDriveRef(stCoE:=HOMS2_YGantry.PAxis.stCoE);
fbInitDriveRef(stCoE:=HOMS2_YGantry.SAxis.stCoE);
fbInitDriveRef(stCoE:=HOMS2_Pitch.Stepper.stCoE);

//Initialze Drive Speeds and Accelerations
//////////////////////////////////////////
HOMS2_XGantry.PAxis.fAcceleration := 1.0;
HOMS2_XGantry.SAxis.fAcceleration := 1.0;
HOMS2_YGantry.PAxis.fAcceleration := 1.0;
HOMS2_YGantry.SAxis.fAcceleration := 1.0;

HOMS2_XGantry.PAxis.fDeceleration := 1.0;
HOMS2_XGantry.SAxis.fDeceleration := 1.0;
HOMS2_YGantry.PAxis.fDeceleration := 1.0;
HOMS2_YGantry.SAxis.fDeceleration := 1.0;

HOMS2_XGantry.PAxis.fVelocity := 0.1;
HOMS2_XGantry.SAxis.fVelocity := 0.1;
HOMS2_YGantry.PAxis.fVelocity := 0.1;
HOMS2_YGantry.SAxis.fVelocity := 0.1;

HOMS2_Pitch.Stepper.fAcceleration := 39;
HOMS2_Pitch.Stepper.fDeceleration := 39;
HOMS2_Pitch.Stepper.fVelocity     := 100;

//Initialize Piezo Driver
/////////////////////////////////////
HOMS2_Pitch.Piezo.stPIParams.fKp := 0.001;
HOMS2_Pitch.Piezo.stPIParams.tTn := T#500MS;
HOMS2_Pitch.Piezo.stPIParams.fOutMaxLimit := 1;
HOMS2_Pitch.Piezo.stPIParams.fOutMinLimit := -1;

// Initialize deadband settings
HOMS2_Pitch.Stepper.rStepperDmovRange := 3;
HOMS2_Pitch.Piezo.rPiezoDmovRange := 0.5;
END_ACTION

ACTION Init_XRTM3:
//FEE-M3
///////////////////////////


//Initialize ELMO Drive references
fbInitDriveRef(stCoE:=HOMS3_XGantry.PAxis.stCoE);
fbInitDriveRef(stCoE:=HOMS3_XGantry.SAxis.stCoE);
fbInitDriveRef(stCoE:=HOMS3_YGantry.PAxis.stCoE);
fbInitDriveRef(stCoE:=HOMS3_YGantry.SAxis.stCoE);
fbInitDriveRef(stCoE:=HOMS3_Pitch.Stepper.stCoE);

//Initialze Drive Speeds and Accelerations
//////////////////////////////////////////
HOMS3_XGantry.PAxis.fAcceleration := 1.0;
HOMS3_XGantry.SAxis.fAcceleration := 1.0;
HOMS3_YGantry.PAxis.fAcceleration := 1.0;
HOMS3_YGantry.SAxis.fAcceleration := 1.0;

HOMS3_XGantry.PAxis.fDeceleration := 1.0;
HOMS3_XGantry.SAxis.fDeceleration := 1.0;
HOMS3_YGantry.PAxis.fDeceleration := 1.0;
HOMS3_YGantry.SAxis.fDeceleration := 1.0;

HOMS3_XGantry.PAxis.fVelocity := 0.1;
HOMS3_XGantry.SAxis.fVelocity := 0.1;
HOMS3_YGantry.PAxis.fVelocity := 0.1;
HOMS3_YGantry.SAxis.fVelocity := 0.1;

HOMS3_Pitch.Stepper.fAcceleration := 39;
HOMS3_Pitch.Stepper.fDeceleration := 39;
HOMS3_Pitch.Stepper.fVelocity     := 100;

//Initialize Piezo Driver
/////////////////////////////////////
HOMS3_Pitch.Piezo.stPIParams.fKp := 0.001;
HOMS3_Pitch.Piezo.stPIParams.tTn := T#500MS;
HOMS3_Pitch.Piezo.stPIParams.fOutMaxLimit := 1;
HOMS3_Pitch.Piezo.stPIParams.fOutMinLimit := -1;

// Initialize deadband settings
HOMS3_Pitch.Stepper.rStepperDmovRange := 20;
HOMS3_Pitch.Piezo.rPiezoDmovRange := 0.5;
END_ACTION

ACTION LimitSwitchIO:
//XRT M2
//////////////////////////
fbM2Y1LS(diInputs:=HOMS2_YGantry.PAxis.diInputs, 
xHiLS=>HOMS2_YGantry.PAxis.xHiLS,
xLoLS=>HOMS2_YGantry.PAxis.xLoLS,
STO => gM2STO);

fbM2Y2LS(diInputs:=HOMS2_YGantry.SAxis.diInputs, 
xHiLS=>HOMS2_YGantry.SAxis.xHiLS,
xLoLS=>HOMS2_YGantry.SAxis.xLoLS);

fbM2X1LS(diInputs:=HOMS2_XGantry.PAxis.diInputs, 
xHiLS=>HOMS2_XGantry.PAxis.xHiLS,
xLoLS=>HOMS2_XGantry.PAxis.xLoLS);

fbM2X2LS(diInputs:=HOMS2_XGantry.SAxis.diInputs, 
xHiLS=>HOMS2_XGantry.SAxis.xHiLS,
xLoLS=>HOMS2_XGantry.SAxis.xLoLS);

fbM2P1LS(Pitch:=HOMS2_Pitch,
xHiLS=>HOMS2_Pitch.Stepper.xHiLS,
xLoLS=>HOMS2_Pitch.Stepper.xLoLS);

//XRT M3
//////////////////////////
fbM3Y1LS(diInputs:=HOMS3_YGantry.PAxis.diInputs, 
xHiLS=>HOMS3_YGantry.PAxis.xHiLS,
xLoLS=>HOMS3_YGantry.PAxis.xLoLS,
STO => gM3STO);

fbM3Y2LS(diInputs:=HOMS3_YGantry.SAxis.diInputs, 
xHiLS=>HOMS3_YGantry.SAxis.xHiLS,
xLoLS=>HOMS3_YGantry.SAxis.xLoLS);

fbM3X1LS(diInputs:=HOMS3_XGantry.PAxis.diInputs, 
xHiLS=>HOMS3_XGantry.PAxis.xHiLS,
xLoLS=>HOMS3_XGantry.PAxis.xLoLS);
(*
fbM3X2LS(diInputs:=HOMS3_XGantry.PAxis.diInputs,  //Paxis is here on purpose <HACK>
xHiLS=>HOMS3_XGantry.SAxis.xHiLS,
xLoLS=>HOMS3_XGantry.SAxis.xLoLS);
*)
fbM3X2LS(diInputs:=HOMS3_XGantry.SAxis.diInputs,  // Switching to SAxis works as expected, reason for <HACK> unclear
xHiLS=>HOMS3_XGantry.SAxis.xHiLS,
xLoLS=>HOMS3_XGantry.SAxis.xLoLS);

fbM3P1LS(Pitch:=HOMS3_Pitch,
xHiLS=>HOMS3_Pitch.Stepper.xHiLS,
xLoLS=>HOMS3_Pitch.Stepper.xLoLS);
END_ACTION

END_PROGRAM

// ---- POUs/Modbus/p_ModbusRx_PLCMemory.TcPOU
PROGRAM p_ModbusRx_PLCMemory
VAR
END_VAR

MEMCPY(srcAddr:=ADR(mb_PLC_Memory[20]), destAddr:=ADR(HOMS2_XGantry.PAxis.rReqAbsolute), n:=SIZEOF(HOMS2_XGantry.PAxis.rReqAbsolute));
MEMCPY(srcAddr:=ADR(mb_PLC_Memory[22]), destAddr:=ADR(HOMS2_XGantry.PAxis.rTweak), n:=SIZEOF(HOMS2_XGantry.PAxis.rTweak));
MEMCPY(srcAddr:=ADR(mb_PLC_Memory[24]), destAddr:=ADR(HOMS2_XGantry.SAxis.rReqAbsolute), n:=SIZEOF(HOMS2_XGantry.SAxis.rReqAbsolute));
MEMCPY(srcAddr:=ADR(mb_PLC_Memory[26]), destAddr:=ADR(HOMS2_XGantry.SAxis.rTweak), n:=SIZEOF(HOMS2_XGantry.SAxis.rTweak));
MEMCPY(srcAddr:=ADR(mb_PLC_Memory[28]), destAddr:=ADR(HOMS2_YGantry.PAxis.rReqAbsolute), n:=SIZEOF(HOMS2_YGantry.PAxis.rReqAbsolute));
MEMCPY(srcAddr:=ADR(mb_PLC_Memory[30]), destAddr:=ADR(HOMS2_YGantry.PAxis.rTweak), n:=SIZEOF(HOMS2_YGantry.PAxis.rTweak));
MEMCPY(srcAddr:=ADR(mb_PLC_Memory[32]), destAddr:=ADR(HOMS2_YGantry.SAxis.rReqAbsolute), n:=SIZEOF(HOMS2_YGantry.SAxis.rReqAbsolute));
MEMCPY(srcAddr:=ADR(mb_PLC_Memory[34]), destAddr:=ADR(HOMS2_YGantry.SAxis.rTweak), n:=SIZEOF(HOMS2_YGantry.SAxis.rTweak));
MEMCPY(srcAddr:=ADR(mb_PLC_Memory[36]), destAddr:=ADR(HOMS2_Pitch.Axis.rReqAbsPos), n:=SIZEOF(HOMS2_Pitch.Axis.rReqAbsPos));
MEMCPY(srcAddr:=ADR(mb_PLC_Memory[38]), destAddr:=ADR(HOMS2_Pitch.Axis.rTweak), n:=SIZEOF(HOMS2_Pitch.Axis.rTweak));
MEMCPY(srcAddr:=ADR(mb_PLC_Memory[40]), destAddr:=ADR(HOMS3_XGantry.PAxis.rReqAbsolute), n:=SIZEOF(HOMS3_XGantry.PAxis.rReqAbsolute));
MEMCPY(srcAddr:=ADR(mb_PLC_Memory[42]), destAddr:=ADR(HOMS3_XGantry.PAxis.rTweak), n:=SIZEOF(HOMS3_XGantry.PAxis.rTweak));
MEMCPY(srcAddr:=ADR(mb_PLC_Memory[44]), destAddr:=ADR(HOMS3_XGantry.SAxis.rReqAbsolute), n:=SIZEOF(HOMS3_XGantry.SAxis.rReqAbsolute));
MEMCPY(srcAddr:=ADR(mb_PLC_Memory[46]), destAddr:=ADR(HOMS3_XGantry.SAxis.rTweak), n:=SIZEOF(HOMS3_XGantry.SAxis.rTweak));
MEMCPY(srcAddr:=ADR(mb_PLC_Memory[48]), destAddr:=ADR(HOMS3_YGantry.PAxis.rReqAbsolute), n:=SIZEOF(HOMS3_YGantry.PAxis.rReqAbsolute));
MEMCPY(srcAddr:=ADR(mb_PLC_Memory[50]), destAddr:=ADR(HOMS3_YGantry.PAxis.rTweak), n:=SIZEOF(HOMS3_YGantry.PAxis.rTweak));
MEMCPY(srcAddr:=ADR(mb_PLC_Memory[52]), destAddr:=ADR(HOMS3_YGantry.SAxis.rReqAbsolute), n:=SIZEOF(HOMS3_YGantry.SAxis.rReqAbsolute));
MEMCPY(srcAddr:=ADR(mb_PLC_Memory[54]), destAddr:=ADR(HOMS3_YGantry.SAxis.rTweak), n:=SIZEOF(HOMS3_YGantry.SAxis.rTweak));
MEMCPY(srcAddr:=ADR(mb_PLC_Memory[56]), destAddr:=ADR(HOMS3_Pitch.Axis.rReqAbsPos), n:=SIZEOF(HOMS3_Pitch.Axis.rReqAbsPos));
MEMCPY(srcAddr:=ADR(mb_PLC_Memory[58]), destAddr:=ADR(HOMS3_Pitch.Axis.rTweak), n:=SIZEOF(HOMS3_Pitch.Stepper.rTweak));

MEMCPY(srcAddr:=ADR(mb_PLC_Memory[64]), destAddr:=ADR(HOMS2_Pitch.Stepper.rStepperDmovRange), n:=SIZEOF(HOMS2_Pitch.Stepper.rStepperDmovRange));
MEMCPY(srcAddr:=ADR(mb_PLC_Memory[66]), destAddr:=ADR(HOMS2_Pitch.Piezo.rPiezoDmovRange), n:=SIZEOF(HOMS2_Pitch.Piezo.rPiezoDmovRange));
MEMCPY(srcAddr:=ADR(mb_PLC_Memory[68]), destAddr:=ADR(HOMS3_Pitch.Stepper.rStepperDmovRange), n:=SIZEOF(HOMS3_Pitch.Stepper.rStepperDmovRange));
MEMCPY(srcAddr:=ADR(mb_PLC_Memory[70]), destAddr:=ADR(HOMS3_Pitch.Piezo.rPiezoDmovRange), n:=SIZEOF(HOMS3_Pitch.Piezo.rPiezoDmovRange));

//MEMCPY(srcAddr:=ADR(mb_PLC_Memory[142]), destAddr:=ADR(HOMS2_Pitch.Piezo.rReqVoltage), n:=SIZEOF(HOMS2_Pitch.Piezo.rReqVoltage));

END_PROGRAM

// ---- POUs/Modbus/p_ModbusTx_PLCMemory.TcPOU
PROGRAM p_ModbusTx_PLCMemory
VAR

END_VAR

MEMCPY(srcAddr:=ADR(HOMS2_XGantry.PAxis.stStatus.rActPosition), destAddr:=ADR(mb_PLC_Memory[130]), n:=SIZEOF(HOMS2_XGantry.PAxis.stStatus.rActPosition));
MEMCPY(srcAddr:=ADR(HOMS2_XGantry.PAxis.stStatus.rActVelocity), destAddr:=ADR(mb_PLC_Memory[132]), n:=SIZEOF(HOMS2_XGantry.PAxis.stStatus.rActVelocity));
MEMCPY(srcAddr:=ADR(HOMS2_XGantry.PAxis.stAxis.NcToPlc.SetAcc), destAddr:=ADR(mb_PLC_Memory[134]), n:=SIZEOF(HOMS2_XGantry.PAxis.stAxis.NcToPlc.SetAcc));
MEMCPY(srcAddr:=ADR(HOMS2_XGantry.SAxis.stStatus.rActPosition), destAddr:=ADR(mb_PLC_Memory[136]), n:=SIZEOF(HOMS2_XGantry.SAxis.stStatus.rActPosition));
MEMCPY(srcAddr:=ADR(HOMS2_XGantry.SAxis.stStatus.rActVelocity), destAddr:=ADR(mb_PLC_Memory[138]), n:=SIZEOF(HOMS2_XGantry.SAxis.stStatus.rActVelocity));
MEMCPY(srcAddr:=ADR(HOMS2_XGantry.SAxis.stAxis.NcToPlc.SetAcc), destAddr:=ADR(mb_PLC_Memory[140]), n:=SIZEOF(HOMS2_XGantry.SAxis.stAxis.NcToPlc.SetAcc));
MEMCPY(srcAddr:=ADR(HOMS2_YGantry.PAxis.stStatus.rActPosition), destAddr:=ADR(mb_PLC_Memory[142]), n:=SIZEOF(HOMS2_YGantry.PAxis.stStatus.rActPosition));
MEMCPY(srcAddr:=ADR(HOMS2_YGantry.PAxis.stStatus.rActVelocity), destAddr:=ADR(mb_PLC_Memory[144]), n:=SIZEOF(HOMS2_YGantry.PAxis.stStatus.rActVelocity));
MEMCPY(srcAddr:=ADR(HOMS2_YGantry.PAxis.stAxis.NcToPlc.SetAcc), destAddr:=ADR(mb_PLC_Memory[146]), n:=SIZEOF(HOMS2_YGantry.PAxis.stAxis.NcToPlc.SetAcc));
MEMCPY(srcAddr:=ADR(HOMS2_YGantry.SAxis.stStatus.rActPosition), destAddr:=ADR(mb_PLC_Memory[148]), n:=SIZEOF(HOMS2_YGantry.SAxis.stStatus.rActPosition));
MEMCPY(srcAddr:=ADR(HOMS2_YGantry.SAxis.stStatus.rActVelocity), destAddr:=ADR(mb_PLC_Memory[150]), n:=SIZEOF(HOMS2_YGantry.SAxis.stStatus.rActVelocity));
MEMCPY(srcAddr:=ADR(HOMS2_YGantry.SAxis.stAxis.NcToPlc.SetAcc), destAddr:=ADR(mb_PLC_Memory[152]), n:=SIZEOF(HOMS2_YGantry.SAxis.stAxis.NcToPlc.SetAcc));
MEMCPY(srcAddr:=ADR(HOMS2_Pitch.Stepper.stStatus.rActPosition), destAddr:=ADR(mb_PLC_Memory[154]), n:=SIZEOF(HOMS2_Pitch.Stepper.stStatus.rActPosition));
MEMCPY(srcAddr:=ADR(HOMS2_Pitch.Stepper.stStatus.rActVelocity), destAddr:=ADR(mb_PLC_Memory[156]), n:=SIZEOF(HOMS2_Pitch.Stepper.stStatus.rActVelocity));
MEMCPY(srcAddr:=ADR(HOMS2_Pitch.Stepper.stAxis.NcToPlc.SetAcc), destAddr:=ADR(mb_PLC_Memory[158]), n:=SIZEOF(HOMS2_Pitch.Stepper.stAxis.NcToPlc.SetAcc));
MEMCPY(srcAddr:=ADR(HOMS2_Pitch.Piezo.rActVoltage), destAddr:=ADR(mb_PLC_Memory[166]), n:=SIZEOF(HOMS2_Pitch.Piezo.rActVoltage));
MEMCPY(srcAddr:=ADR(HOMS2_Pitch.Piezo.UpperVoltage), destAddr:=ADR(mb_PLC_Memory[168]), n:=SIZEOF(HOMS2_Pitch.Piezo.UpperVoltage));
MEMCPY(srcAddr:=ADR(HOMS2_Pitch.Piezo.LowerVoltage), destAddr:=ADR(mb_PLC_Memory[170]), n:=SIZEOF(HOMS2_Pitch.Piezo.LowerVoltage));
MEMCPY(srcAddr:=ADR(HOMS2_XGantry.DiffTol), destAddr:=ADR(mb_PLC_Memory[180]), n:=SIZEOF(HOMS2_XGantry.DiffTol));
MEMCPY(srcAddr:=ADR(HOMS2_XGantry.Diff), destAddr:=ADR(mb_PLC_Memory[182]), n:=SIZEOF(HOMS2_XGantry.Diff));
MEMCPY(srcAddr:=ADR(HOMS2_YGantry.DiffTol), destAddr:=ADR(mb_PLC_Memory[184]), n:=SIZEOF(HOMS2_YGantry.DiffTol));
MEMCPY(srcAddr:=ADR(HOMS2_YGantry.Diff), destAddr:=ADR(mb_PLC_Memory[186]), n:=SIZEOF(HOMS2_YGantry.Diff));



MEMCPY(destAddr:=ADR(mb_PLC_Memory[36]), srcAddr:=ADR(HOMS2_Pitch.Axis.rReqAbsPos), n:=SIZEOF(HOMS2_Pitch.Axis.rReqAbsPos));
MEMCPY(destAddr:=ADR(mb_PLC_Memory[56]), srcAddr:=ADR(HOMS3_Pitch.Axis.rReqAbsPos), n:=SIZEOF(HOMS3_Pitch.Axis.rReqAbsPos));

MEMCPY(srcAddr:=ADR(HOMS3_XGantry.PAxis.stStatus.rActPosition), destAddr:=ADR(mb_PLC_Memory[188]), n:=SIZEOF(HOMS3_XGantry.PAxis.stStatus.rActPosition));
MEMCPY(srcAddr:=ADR(HOMS3_XGantry.PAxis.stStatus.rActVelocity), destAddr:=ADR(mb_PLC_Memory[190]), n:=SIZEOF(HOMS3_XGantry.PAxis.stStatus.rActVelocity));
MEMCPY(srcAddr:=ADR(HOMS3_XGantry.PAxis.stAxis.NcToPlc.SetAcc), destAddr:=ADR(mb_PLC_Memory[192]), n:=SIZEOF(HOMS3_XGantry.PAxis.stAxis.NcToPlc.SetAcc));
MEMCPY(srcAddr:=ADR(HOMS3_XGantry.SAxis.stStatus.rActPosition), destAddr:=ADR(mb_PLC_Memory[194]), n:=SIZEOF(HOMS3_XGantry.SAxis.stStatus.rActPosition));
MEMCPY(srcAddr:=ADR(HOMS3_XGantry.SAxis.stStatus.rActVelocity), destAddr:=ADR(mb_PLC_Memory[196]), n:=SIZEOF(HOMS3_XGantry.SAxis.stStatus.rActVelocity));
MEMCPY(srcAddr:=ADR(HOMS3_XGantry.SAxis.stAxis.NcToPlc.SetAcc), destAddr:=ADR(mb_PLC_Memory[198]), n:=SIZEOF(HOMS3_XGantry.SAxis.stAxis.NcToPlc.SetAcc));
MEMCPY(srcAddr:=ADR(HOMS3_YGantry.PAxis.stStatus.rActPosition), destAddr:=ADR(mb_PLC_Memory[200]), n:=SIZEOF(HOMS3_YGantry.PAxis.stStatus.rActPosition));
MEMCPY(srcAddr:=ADR(HOMS3_YGantry.PAxis.stStatus.rActVelocity), destAddr:=ADR(mb_PLC_Memory[202]), n:=SIZEOF(HOMS3_YGantry.PAxis.stStatus.rActVelocity));
MEMCPY(srcAddr:=ADR(HOMS3_YGantry.PAxis.stAxis.NcToPlc.SetAcc), destAddr:=ADR(mb_PLC_Memory[204]), n:=SIZEOF(HOMS3_YGantry.PAxis.stAxis.NcToPlc.SetAcc));
MEMCPY(srcAddr:=ADR(HOMS3_YGantry.SAxis.stStatus.rActPosition), destAddr:=ADR(mb_PLC_Memory[206]), n:=SIZEOF(HOMS3_YGantry.SAxis.stStatus.rActPosition));
MEMCPY(srcAddr:=ADR(HOMS3_YGantry.SAxis.stStatus.rActVelocity), destAddr:=ADR(mb_PLC_Memory[208]), n:=SIZEOF(HOMS3_YGantry.SAxis.stStatus.rActVelocity));
MEMCPY(srcAddr:=ADR(HOMS3_YGantry.SAxis.stAxis.NcToPlc.SetAcc), destAddr:=ADR(mb_PLC_Memory[210]), n:=SIZEOF(HOMS3_YGantry.SAxis.stAxis.NcToPlc.SetAcc));
MEMCPY(srcAddr:=ADR(HOMS3_Pitch.Stepper.stStatus.rActPosition), destAddr:=ADR(mb_PLC_Memory[212]), n:=SIZEOF(HOMS3_Pitch.Stepper.stStatus.rActPosition));
MEMCPY(srcAddr:=ADR(HOMS3_Pitch.Stepper.stStatus.rActVelocity), destAddr:=ADR(mb_PLC_Memory[214]), n:=SIZEOF(HOMS3_Pitch.Stepper.stStatus.rActVelocity));
MEMCPY(srcAddr:=ADR(HOMS3_Pitch.Stepper.stAxis.NcToPlc.SetAcc), destAddr:=ADR(mb_PLC_Memory[216]), n:=SIZEOF(HOMS3_Pitch.Stepper.stAxis.NcToPlc.SetAcc));
MEMCPY(srcAddr:=ADR(HOMS3_Pitch.Piezo.rActVoltage), destAddr:=ADR(mb_PLC_Memory[218]), n:=SIZEOF(HOMS3_Pitch.Piezo.rActVoltage));
MEMCPY(srcAddr:=ADR(HOMS3_Pitch.Piezo.UpperVoltage), destAddr:=ADR(mb_PLC_Memory[220]), n:=SIZEOF(HOMS3_Pitch.Piezo.UpperVoltage));
MEMCPY(srcAddr:=ADR(HOMS3_Pitch.Piezo.LowerVoltage), destAddr:=ADR(mb_PLC_Memory[222]), n:=SIZEOF(HOMS3_Pitch.Piezo.LowerVoltage));
MEMCPY(srcAddr:=ADR(HOMS3_XGantry.DiffTol), destAddr:=ADR(mb_PLC_Memory[224]), n:=SIZEOF(HOMS3_XGantry.DiffTol));
MEMCPY(srcAddr:=ADR(HOMS3_XGantry.Diff), destAddr:=ADR(mb_PLC_Memory[226]), n:=SIZEOF(HOMS3_XGantry.Diff));
MEMCPY(srcAddr:=ADR(HOMS3_YGantry.DiffTol), destAddr:=ADR(mb_PLC_Memory[228]), n:=SIZEOF(HOMS3_YGantry.DiffTol));
MEMCPY(srcAddr:=ADR(HOMS3_YGantry.Diff), destAddr:=ADR(mb_PLC_Memory[230]), n:=SIZEOF(HOMS3_YGantry.Diff));

MEMCPY(srcAddr:=ADR(HOMS2_Pitch.ReqPosLimLo), destAddr:=ADR(mb_PLC_Memory[236]), n:=SIZEOF(HOMS2_Pitch.ReqPosLimLo));
MEMCPY(srcAddr:=ADR(HOMS2_Pitch.ReqPosLimHi), destAddr:=ADR(mb_PLC_Memory[238]), n:=SIZEOF(HOMS2_Pitch.ReqPosLimHi));
MEMCPY(srcAddr:=ADR(HOMS3_Pitch.ReqPosLimLo), destAddr:=ADR(mb_PLC_Memory[240]), n:=SIZEOF(HOMS3_Pitch.ReqPosLimLo));
MEMCPY(srcAddr:=ADR(HOMS3_Pitch.ReqPosLimHi), destAddr:=ADR(mb_PLC_Memory[242]), n:=SIZEOF(HOMS3_Pitch.ReqPosLimHi));

MEMCPY(destAddr:=ADR(mb_PLC_Memory[64]), srcAddr:=ADR(HOMS2_Pitch.Stepper.rStepperDmovRange), n:=SIZEOF(HOMS2_Pitch.Stepper.rStepperDmovRange));
MEMCPY(destAddr:=ADR(mb_PLC_Memory[66]), srcAddr:=ADR(HOMS2_Pitch.Piezo.rPiezoDmovRange), n:=SIZEOF(HOMS2_Pitch.Piezo.rPiezoDmovRange));
MEMCPY(destAddr:=ADR(mb_PLC_Memory[68]), srcAddr:=ADR(HOMS3_Pitch.Stepper.rStepperDmovRange), n:=SIZEOF(HOMS3_Pitch.Stepper.rStepperDmovRange));
MEMCPY(destAddr:=ADR(mb_PLC_Memory[70]), srcAddr:=ADR(HOMS3_Pitch.Piezo.rPiezoDmovRange), n:=SIZEOF(HOMS3_Pitch.Piezo.rPiezoDmovRange));


//MEMCPY(destAddr:=ADR(mb_PLC_Memory[256]), srcAddr:=ADR(HOMS3_Pitch.Axis.rReqAbsPos), n:=SIZEOF(HOMS3_Pitch.Stepper.rReqAbsolute));

END_PROGRAM

// ---- POUs/PRG_CoatingProtection.TcPOU
PROGRAM PRG_CoatingProtection
VAR
	//M1 
   fbM1 : FB_MirrorCoatingProtection := (
	   	sDevName:= 'XRT-M1', 
		rFirstCoatingPosition:= 8611000, 
		rFirstCoatingPositionTolerance:= 1000000, 
		nFirstCoatingBitmask:= 2#0000_0001_1111_1111, 
		sFirstCoatingType:= 'SiC', 
		rSecondCoatingPosition:= 18611000 , 
		rSecondCoatingPositionTolerance:= 1000000 , 
		nSecondCoatingBitmask:=  2#1111_1100_0000_0000 , 
		sSecondCoatingType:= 'W', 
		bAutoClear:= TRUE);
		

//M2
   fbM2 : FB_MirrorCoatingProtection := (
	   	sDevName:= 'XRT-M2', 
		rFirstCoatingPosition:= 8496030, 
		rFirstCoatingPositionTolerance:= 1000000, 
		sFirstCoatingType:= 'SiC', 
		rSecondCoatingPosition:= 18496030 , 
		rSecondCoatingPositionTolerance:= 1000000 , 
		sSecondCoatingType:= 'W', 
		bAutoClear:= TRUE);

		
//M3 
   fbM3 : FB_MirrorCoatingProtection := (
	   	sDevName:= 'XRT-M3', 
		rFirstCoatingPosition:= 9279350, 
		rFirstCoatingPositionTolerance:= 1000000, 
		nFirstCoatingBitmask:= 2#0000_0001_1111_1111, 
		sFirstCoatingType:= 'SiC', 
		rSecondCoatingPosition:= 19279350 , 
		rSecondCoatingPositionTolerance:= 1000000 , 
		nSecondCoatingBitmask:=  2#1111_1100_0000_0000 , 
		sSecondCoatingType:= 'W', 
		bAutoClear:= TRUE);		
	
		//PMPS arbiter Interface
		fbArbiterIO : FB_SubSysToArbiter_IO;
		rtRemove: R_TRIG;
		bRemove :BOOL;
		bExist :BOOL;
		nReq : UDINT;
		
           
END_VAR


//M1
fbM1(
	bMirrorIn := (Main.nEncCntXupXRTM1 > 20210500) , // according to confluence -6 is nominal out position
    rCurrentEncoderPosition := Main.nEncCntYupXRTM1,
    neVRange := PMPS.PMPS_GVL.stCurrentBeamParameters.neVRange,
    FFO := GVL_PMPS.g_FastFaultOutput1);
	
//M2
//With M2 the same coating has different bit masks depending on the pitch
IF (HOMS2_Pitch.diEncCnt < 9616668 ) THEN//(HOMS2_Pitch.Stepper.stStatus.rActPosition < -400 ) THEN //MFX
	fbM2.nFirstCoatingBitmask:= 2#0000_0001_1111_1111; 
	fbM2.nSecondCoatingBitmask:= 2#1111_1100_0000_0000; 
ELSIF (HOMS2_Pitch.diEncCnt > 10129409 ) THEN// (HOMS2_Pitch.Stepper.stStatus.rActPosition > 600) THEN //MEC
	fbM2.nFirstCoatingBitmask:= 2#1111_1111_1111_1111;  
	fbM2.nSecondCoatingBitmask:= 2#1111_1100_0000_0000;  
ELSE // Anything else in the middle of the range
	fbM2.nFirstCoatingBitmask:= 2#0000_0000_0000_0000; 
	fbM2.nSecondCoatingBitmask:= 2#0000_0000_0000_0000;  		
END_IF

fbM2(
	bMirrorIn := (HOMS2_XGantry.PAxis.diEncCnt < 25490840), 
    rCurrentEncoderPosition := HOMS2_YGantry.PAxis.diEncCnt,
    neVRange := PMPS.PMPS_GVL.stCurrentBeamParameters.neVRange,
    FFO := GVL_PMPS.g_FastFaultOutput1);

	
//M3
fbM3(
	bMirrorIn:=  fbM1.bMirrorIn, // When M1 is out, M3 is considered to be OUT
    rCurrentEncoderPosition := HOMS3_YGantry.PAxis.diEncCnt,
    neVRange := PMPS.PMPS_GVL.stCurrentBeamParameters.neVRange,
    FFO := GVL_PMPS.g_FastFaultOutput1);
	
	
// PMPS ARbiter and FFO instantiation.
GVL_PMPS.g_fbArbiter1.AddRequest(16#5, PMPS_GVL.cstFullBeam);
fbArbiterIO(Arbiter := GVL_PMPS.g_fbArbiter1, fbFFHWO := GVL_PMPS.g_FastFaultOutput1);
GVL_PMPS.g_FastFaultOutput1.Execute(bAutoReset:=TRUE, i_xVeto:=);
GVL_PMPS.g_FastFaultOutput2.Execute(bAutoReset:=TRUE, i_xVeto:=);	

bExist:= GVL_PMPS.g_fbArbiter1.CheckRequestInPool(nReq);
rtRemove(CLK:= bRemove);
if (rtRemove.Q) THEN
 	GVL_PMPS.g_fbArbiter1.RemoveRequest(nReq); 
END_IF

END_PROGRAM

// ---- POUs/Serial Comm/PiezoSerial.TcPOU
PROGRAM PiezoSerial
VAR
	//PI Serial
	fbE621SerialDriverM1 : FB_PI_E621_SerialDriver;
	fbE621SerialDriverM2 : FB_PI_E621_SerialDriver;
	fbE621SerialDriverM3 : FB_PI_E621_SerialDriver;
	rtInitParams	:	R_TRIG;
	tonTimeoutRstM1	: TON := (PT:=T#2S); //For timeout reset
	tonTimeoutRstM2	: TON := (PT:=T#2S); //For timeout reset
END_VAR

//M1 Piezo E-621
///////////////////////
	fbE621SerialDriverM1.i_xExecute := TRUE;
	fbE621SerialDriverM1.i_xExecute R= fbE621SerialDriverM1.q_xDone;
	fbE621SerialDriverM1(
		iq_stPiezoAxis:= GVL_XRTM1.XRTM1_Pitch.Piezo, 
		iq_stSerialRXBuffer:= Serial_P1_SerialRXBuffer, 
		iq_stSerialTXBuffer:= Serial_P1_SerialTXBuffer);
	
//M2 Piezo E-621
///////////////////////
	fbE621SerialDriverM2.i_xExecute := TRUE;
	fbE621SerialDriverM2.i_xExecute R= fbE621SerialDriverM2.q_xDone;
	fbE621SerialDriverM2(
		iq_stPiezoAxis:= HOMS2_Pitch.Piezo, 
		iq_stSerialRXBuffer:= Serial_P2_SerialRXBuffer, 
		iq_stSerialTXBuffer:= Serial_P2_SerialTXBuffer);
		
//M3 Piezo E-621
///////////////////////
	fbE621SerialDriverM3.i_xExecute := TRUE;
	fbE621SerialDriverM3.i_xExecute R= fbE621SerialDriverM3.q_xDone;
	fbE621SerialDriverM3(
		iq_stPiezoAxis:= HOMS3_Pitch.Piezo, 
		iq_stSerialRXBuffer:= Serial_P3_SerialRXBuffer, 
		iq_stSerialTXBuffer:= Serial_P3_SerialTXBuffer);

END_PROGRAM
